FUNCTION alg_a_HledQ1 : BOOL
VAR_INPUT
	state: STATE;
END_VAR

alg_a_HledQ1 := FALSE;

END_FUNCTION

(* stored: Version 1.1.0.1, ProductVersion 3.1.4022.18
   POU alg_a_HledQ1: Id {272121cc-6e76-4773-bcd0-1559d82a151c}, SpecialFunc None *)
